PROPERTY WareHouseClampA_Handshake : ST_Fanuc_WarehouseHandshake
GET
WareHouseClampA_Handshake := _DO1;
END_GET
SET
// Outside -> FB 
_DO1 := WareHouseClampA_Handshake;
END_SET
END_PROPERTY

PROPERTY WareHouseClampB_Handshake : ST_Fanuc_WarehouseHandshake
GET
WareHouseClampB_Handshake := _DO2;
END_GET
SET
// Outside -> FB 
_DO2 := WareHouseClampB_Handshake;
END_SET
END_PROPERTY

PROPERTY Write_OffsetP : INT
SET
_DI11 := Write_OffsetP;
END_SET
END_PROPERTY

PROPERTY Write_OffsetR : INT
SET
_DO12 := Write_OffsetR;
END_SET
END_PROPERTY

PROPERTY Write_OffsetW : INT
SET
_DO10 := Write_OffsetW;
END_SET
END_PROPERTY

PROPERTY Write_OffsetX : INT
SET
_DO7 := Write_OffsetX;
END_SET
END_PROPERTY

PROPERTY Write_OffsetY : INT
SET
_DO8 := Write_OffsetY;
END_SET
END_PROPERTY

PROPERTY Write_OffsetZ : INT
SET
_DO9 := Write_OffsetZ;
END_SET
END_PROPERTY

PROPERTY WriteDataCommand : bool;
SET
_DO6.WritePara_Execute := WriteDataCommand;
END_SET
END_PROPERTY

END_FUNCTION_BLOCK

(* stored: Version 1.1.0.1, ProductVersion 3.1.4024.13
   POU FB_FanucRobot_Basic_V2: Id {cb73f1fe-6ec3-4c6c-8f86-ed9d19b8966c}, SpecialFunc None
   Folder Action: Id {cb276f10-ba0c-420d-b693-c3ed88186172}
   Folder HandShake: Id {e1dea49a-519d-4068-a110-3f88453f47a2}
   Folder Method: Id {56c3ffc1-bb0d-4ffc-a087-cdf2b0bfa324}
   Folder ManualService: Id {8e48eb1a-a1e8-4853-8878-cc3a05fa7e55}
   Folder ModeControl: Id {4f814264-21dc-4148-978f-a27c3702b438}
   Folder MoveBoxToFeedInConveyor: Id {c9d6e2f9-e9a0-4b89-852b-cc310f8857b3}
   Folder MoveBoxToRoundBelt: Id {6b98bebc-f19a-4f6a-a41d-27031a7739e4}
   Folder PickBoxFromRoundBelt: Id {676c8d97-f52e-4807-87ad-dec847256722}
   Folder PulloutConveyor PickupBox: Id {54747d94-7097-47ed-86d5-04c2c29ec3a8}
   Folder RobotAbsMove: Id {fca1ac7b-8fd2-4c25-a683-c608de9a23a8}
   Folder RobotAction: Id {8edbc682-62f4-44bc-b4cb-0bd7b86f9e10}
   Folder Reset: Id {a74a37e1-3a7a-4b93-b002-be43b29154c4}
   Folder ShippingRobotAction: Id {099c541b-ccb7-4755-84de-e892f4455303}
   Folder Warehouse PickupBox: Id {e5de1fd4-e1a6-44f8-8306-7a04a63b9506}
   Folder Warehouse PlaceBox: Id {9aff1c5b-54a4-4f10-aca8-eb5391878d40}
   Action A00_BaseUnit: Id {1f9035bb-8d05-4b96-8e6d-aa3ad82503cc}
   Action A10_ModeControl: Id {f8257065-0214-442d-a7cb-43b8b0292644}
   Action A20_ErrorHandle: Id {c7f664ad-e2ac-4eb6-8e44-2a0d78101723}
   Action A20_StateControl: Id {c464481d-37e5-4287-aded-0f09353e249c}
   Property AbsMoveClampA_Handshake: Id {c2b1fd16-5fce-4025-adcc-2ab9b488ab57}
   Get Get: Id {fd93046e-8d52-455f-b85c-a592225045f9}
   Set Set: Id {85a7ea43-512b-4f2b-9ceb-eaae03b35005}
   Property AbsMoveClampB_Handshake: Id {bca207b7-83c6-433d-a7ec-6f4e9cc2a310}
   Get Get: Id {1c5120ba-971a-42a0-b47f-a9695f0fd70f}
   Set Set: Id {07a5d79e-2714-455e-b0bf-a38889d531fc}
   Property Bzone_AllowWork: Id {9f8f4c55-d2a2-4ab8-91c2-d0bc6074ba44}
   Get Get: Id {6ccc57ff-b0e6-4950-9dfa-51cf4d4323d7}
   Set Set: Id {8d47b4d6-2402-4629-aefe-2f1bbce98ca4}
   Property BZoneInWork: Id {6071e1db-41bd-4366-8b7f-cda085c54340}
   Get Get: Id {d85d4e07-ceaa-44ab-89cf-0c6fde819275}
   Property Command: Id {7b43bc35-fea1-4857-98a1-06622f0ea970}
   Get Get: Id {19c06e74-acc7-4709-aaeb-6891ab645997}
   Set Set: Id {e54317f6-93a0-424d-b6e6-9398ae0f1ca3}
   Method Enable: Id {d6452130-06a4-4b03-9e85-1071184db1ab}
   Method EStop: Id {d0568f40-b052-42be-a0f8-d45c1a9b95a7}
   Property FanucRobot_MotionStatus: Id {5f69344f-7f0a-4846-9adc-c1a5e377b175}
   Get Get: Id {c8f5df37-a69d-4e0c-8408-22ea6f345c3f}
   Method Fault: Id {5786630b-c79e-45db-abf4-bb0ce3df87fc}
   Method GetModelState: Id {84684909-97c4-4c1d-88c5-578deecdb205}
   Method GetName: Id {286e5c35-9036-4531-9db3-ece6debb9b2d}
   Method Hold: Id {1474dcf7-848d-4116-a653-f29314484d4e}
   Property Homed: Id {d2ee59f6-70a7-4539-818a-3e783665ccea}
   Get Get: Id {b8cf7904-7492-4902-bccd-4143cae76aee}
   Property LayerIndex: Id {ef35ac31-f7e6-4395-8b6b-894321314b34}
   Set Set: Id {cf4e2c21-c483-4e00-b34a-37a3bcb4c4f9}
   Method M_ActiveRSR01: Id {c552c3cd-353a-47d5-89f3-e9c40429c882}
   Method M_ActiveRSR02: Id {852e35c1-33f2-4795-83cd-808f6b0ff594}
   Method M_ActiveRSR03: Id {b3fc9105-3a60-403e-b13b-10e04e5bab64}
   Method M_CheckResetAllCommand: Id {4f0eeb7c-ae1a-4f02-8479-69d5b6e0d8de}
   Method M_ClearState: Id {1952fa3e-6dba-4673-9d16-d8027aada721}
   Method M_ControlRSR01: Id {bcb4fe96-4792-4404-912c-6714ffc321c9}
   Method M_ControlRSR02: Id {8e129eae-e0be-4da0-a048-edee41293866}
   Method M_ControlRSR03: Id {83abdd3b-2b3b-4c43-85dc-c5894cb7ff45}
   Method M_EnableWith4Input: Id {657ee152-aee4-4b2b-ae77-0fafc788075b}
   Method M_GetErrorCode: Id {1faf4c23-25ec-44cf-8d8d-0bffb575c5e7}
   Method M_Kawasaki_API: Id {a99effd1-dac7-4001-a6a2-2106ed5eb6cc}
   Method M_ManualService: Id {2546a455-5a0b-40b7-b479-3a695cf9c66f}
   Method M_ReleaseRobotInternalCycle: Id {021b4c72-90a6-425c-a65b-affa6c1b2330}
   Method M_Reset: Id {d945901e-d9fe-42ce-8de4-ab43b85fae1b}
   Method M_ResetAbsMoveClampACommand: Id {7adf9837-6458-4204-9144-b1ea423e4711}
   Method M_ResetAbsMoveClampBCommand: Id {7e76b191-79e1-4364-8390-d69576d859d6}
   Method M_ResetAbsMoveCommand: Id {90b9405a-693f-4171-81c8-3ba8eb66b7f3}
   Method M_ResetAllCommand: Id {e917d518-47fb-4c39-90c3-2a2c59c2fa61}
   Method M_ResetInternalCycleCommand: Id {1e8bf53f-2251-4e1a-8199-4992392cbf0c}
   Method M_ResetMoveBoxToFeedInConveyor_ClampA: Id {3fdff994-4c03-410e-8b67-0a65dd7ab89c}
   Method M_ResetMoveBoxToFeedInConveyor_ClampB: Id {a95c3a8e-845d-4f0f-b2f4-c51448ed0bbe}
   Method M_ResetMoveBoxToFeedInConveyor_ClampBoth: Id {9216c864-92f3-4422-85fa-6b22bd94d3e0}
   Method M_ResetMoveBoxToRoundBelt_Both: Id {982ccaa3-7fb1-47b0-9f35-7f6373b184f3}
   Method M_ResetPullOutConveyorPickUpBox_ClampA: Id {2bc954db-3c72-41d5-bd86-6f9fda7a7d49}
   Method M_ResetPullOutConveyorPickUpBox_ClampB: Id {673746db-f506-4a79-acbe-07dc6f4c2208}
   Method M_ResetPullOutConveyorPickUpBox_ClampBoth: Id {6ea528ea-9f24-4d05-a052-7dd240231e93}
   Method M_ResetRobotAbsMove: Id {ae3d86ba-d954-4f18-a3d7-5aff984d30d4}
   Method M_ResetWareHouseClampACommand: Id {8c225284-c6e2-4835-836c-cbf110de026e}
   Method M_ResetWareHouseClampBCommand: Id {055aa34d-cede-4533-adee-7bcb7c644b78}
   Method M_ResetWareHouseCommand: Id {c52f891b-c018-4c95-a75f-1c34a3dfd3fb}
   Method M_ResetWareHousePickUpBox_ClampA: Id {272ffa04-cb30-4f78-be5d-9530710016f7}
   Method M_ResetWareHousePickUpBox_ClampB: Id {6c3f7292-7554-421c-b337-c0d0d72f2903}
   Method M_ResetWareHousePickUpBox_ClampBoth: Id {29756699-b61c-4725-a7be-b048802eede3}
   Method M_StartAbsMoveAction_ClampA: Id {7ee5f088-fcc4-4816-9cbc-e4b5808f6396}
   Method M_StartAbsMoveAction_ClampB: Id {7f2e6fb2-5682-4183-bff8-79d648b497b8}
   Method M_StartAbsMoveAction_ClampBoth: Id {a1efb706-d769-4056-8872-70cad6ae74b3}
   Method M_StartMoveBoxToFeedInConveyor_ClampA: Id {8cc75a07-61c8-44dc-8ea1-497d46928096}
   Method M_StartMoveBoxToFeedInConveyor_ClampB: Id {67597b53-3184-4c3c-b945-b7e9ad582fcd}
   Method M_StartMoveBoxToFeedInConveyor_ClampBoth: Id {1f893b1b-487d-4898-974d-4f2ea9c3b8ae}
   Method M_StartMoveBoxToRoundBelt_Both: Id {7033ebf4-512e-4629-9b48-8880af596849}
   Method M_StartMoveBoxToRoundBelt_ClampA: Id {b5b94ab9-c903-453f-8523-025cde3b628b}
   Method M_StartMoveBoxToRoundBelt_ClampB: Id {7aeb67a5-dd02-4488-ba5f-e0767b3381ba}
   Method M_StartPickBoxFromRoundBelt_ClampA: Id {029fdc09-38a6-4e13-a6ce-a71c0377098e}
   Method M_StartPickBoxFromRoundBelt_ClampB: Id {bf9c313d-22c3-45b5-8988-5d354c26b927}
   Method M_StartPullOutConveyorPickUpBox_ClampA: Id {55d65623-5d4f-41b7-ad7b-2170591d4a63}
   Method M_StartPullOutConveyorPickUpBox_ClampB: Id {6174b422-22f1-4411-80c3-10a8e781346b}
   Method M_StartPullOutConveyorPickUpBox_ClampBoth: Id {47d1d672-94f3-4ba5-8fdb-d4203337a3ca}
   Method M_StartRobotAbsMove: Id {e8182768-4f43-4df3-8649-d8375ff7bfa3}
   Method M_StartWarehouseMoveAction_ClampA: Id {74d1545f-60b6-4bf2-a234-ebc4eb44d948}
   Method M_StartWarehouseMoveAction_ClampB: Id {a3258f00-624f-45b7-a312-9dff3c52d01d}
   Method M_StartWarehouseMoveAction_ClampBoth: Id {25ac45a8-260f-4e8c-b0dc-4941daaed16e}
   Method M_StartWareHousePickUpBox_ClampA: Id {a175544f-ba2c-498f-8e86-b0560adb92a4}
   Method M_StartWareHousePickUpBox_ClampB: Id {b78797d2-43c2-4f32-8d5c-9bca3fa57483}
   Method M_StartWareHousePickUpBox_ClampBoth: Id {36382dda-f692-4f56-a9ce-af666abd28b8}
   Method M_StartWareHousePlaceBox_ClampA: Id {d7deb918-b191-4624-ab52-b7d9a5a96473}
   Method M_StartWareHousePlaceBox_ClampB: Id {e7972c25-d33e-4f85-9bc8-545c9cc685b6}
   Method M_StartWareHousePlaceUpBox_ClampBoth: Id {b5b211dd-f3f8-473c-8138-2418c6b41ef0}
   Method M_SwitchRSR3: Id {bb1030da-fb99-468b-b550-bf4ad5470872}
   Property Read_OffsetP: Id {4b2241dc-b507-4112-9f01-cd03b33d16b7}
   Get Get: Id {a08568d2-5129-45b0-9f98-d0920c87c238}
   Property Read_OffsetR: Id {6d718848-2859-4b45-9b6a-9d5b1c28f3d7}
   Get Get: Id {0b8f889b-9233-43c2-9ff0-51a13582bbae}
   Property Read_OffsetW: Id {4b83dc30-e29c-4659-b896-51f94a7ea8fe}
   Get Get: Id {8af08794-6483-4d60-87a6-41e7588ead4f}
   Property Read_OffsetX: Id {ec80bea9-7cb9-4e87-a170-a11b11f29db1}
   Get Get: Id {cf3f2d37-b410-4577-ae14-1f6935c5c739}
   Property Read_OffsetY: Id {92f5b32d-2077-4649-b8d3-4e1fdd82d7f6}
   Get Get: Id {eac2a901-17d1-48ca-b77d-174050879008}
   Property Read_OffsetZ: Id {636ddf91-f721-4c7d-b6fc-c5f70aa2544d}
   Get Get: Id {353bca95-e3b0-4040-aa5b-cd7500d0a9e5}
   Property ReadDataCommand: Id {679e0ffa-0848-43b8-99e6-1dd32e72c10a}
   Set Set: Id {d05b65ee-81d9-4ce6-8213-107ac7f16285}
   Property ReadWrite_Address: Id {90b0f67e-f41a-49c5-887c-f46aea83f2ea}
   Set Set: Id {58ac0610-93da-4822-accc-2f457505b187}
   Property ReadWrite_Area: Id {4a6ef189-8220-4f9c-897c-e6934abbeedd}
   Set Set: Id {e28a2607-7b16-41e8-91c1-265de32a2fbe}
   Property ReadWrite_ClampA: Id {12b1eeb8-b518-4284-88b8-83ec160bf71c}
   Set Set: Id {d64441c9-3b45-4c72-94a7-9fa7c1783bc6}
   Property ReadWrite_ClampB: Id {1f63e153-92d1-4676-8d72-c71b9e23a418}
   Set Set: Id {855c2f58-018f-40d0-b34b-adebba39f389}
   Property ReadWrite_WareHouseA: Id {02c81392-db5f-44c7-9b93-e4e044b734ee}
   Set Set: Id {e9ac02ca-849a-48c4-a183-016b6acf8971}
   Property ReadWrite_WareHouseB: Id {4f812627-2f21-4d09-80e8-bd24cf7501a5}
   Set Set: Id {285bfe4e-54e0-4650-99d7-8fdf095b72c5}
   Property ReadyOperation: Id {c6fa2556-761e-4dc3-8374-6e28e08fd2ad}
   Get Get: Id {e3737b9c-783e-47dc-8776-9719123ddaab}
   Property ReadySetParameter: Id {91257f81-5c20-4914-86a7-a3dfaf66b0cd}
   Get Get: Id {f3faab59-a388-4337-9c1a-202df640cb8d}
   Method ReBoot: Id {94db228b-0f78-4766-8c22-25eab32d305c}
   Property SlideIndex: Id {03e8a0af-5644-434f-a0fb-3f3e7ac08bdd}
   Set Set: Id {db45a197-7bfa-4d02-8570-f192d5d9d9be}
   Property Status: Id {ccf81927-043d-434c-9f2d-0605c0f6abc2}
   Get Get: Id {34501a67-89c8-465a-b238-38c5b4605ac6}
   Method Update: Id {3a192417-bff9-4b83-9ccf-83729fdd2006}
   Property VelocityCommand: Id {18bc1b8b-1af2-4445-8cb6-fa03434fba71}
   Get Get: Id {aa359086-9a5f-4772-ba2f-2588e0c2846d}
   Set Set: Id {bf09e38a-58c3-4ecd-b50f-7640ddd22136}
   Property WareHouseClampA_Handshake: Id {f8f665a9-3cba-4c23-9593-852234907303}
   Get Get: Id {125366c5-76b3-40ab-bf1e-165547ab4be8}
   Set Set: Id {b5231219-468f-4fc0-8e7a-fd9b2ab1e073}
   Property WareHouseClampB_Handshake: Id {b1f35835-42cb-46aa-b0b9-91164b8adb3b}
   Get Get: Id {1fe48030-d663-46c9-9e7a-f685a596f201}
   Set Set: Id {83f388e7-54bc-4036-ac28-d75534fd2482}
   Property Write_OffsetP: Id {4daf472e-6895-4e8a-a85c-5248c3789280}
   Set Set: Id {11e0bd42-bc66-4d20-ab51-9601b04a2aa2}
   Property Write_OffsetR: Id {91579b74-f40b-4aae-9c5a-9bee56116c2e}
   Set Set: Id {b8263851-6bcc-4c0f-ba53-cc59703e3b7f}
   Property Write_OffsetW: Id {0781e96b-eca7-479a-a1c5-70f379acc589}
   Set Set: Id {17952dee-7a5e-4fb9-a9d3-a8288c4f86a1}
   Property Write_OffsetX: Id {d113acca-12dd-43cd-a8c7-572ecc9eb398}
   Set Set: Id {5fef888a-263a-4eaf-bf2a-61465ec26c96}
   Property Write_OffsetY: Id {ad026816-e7f0-48ea-a52a-3c41f873dddb}
   Set Set: Id {767f8d1c-2ee2-4469-9338-6540f5e4b04b}
   Property Write_OffsetZ: Id {d3a7f6fb-c026-4022-a46e-104fc8326ec8}
   Set Set: Id {9f002b72-29bd-4d29-a419-5cdd2db1ce3d}
   Property WriteDataCommand: Id {18159747-f74e-4014-84bd-4700b6198c3b}
   Set Set: Id {9b298a4a-6699-48a0-8f74-519aadd6825e} *)
